// TIA Portal V18 export
DATA_BLOCK "AXIS_Y_Motion_V2_Festo_PtP_Drives_PN_DB"   // DB1
AUTHOR : Festo
FAMILY : E-.Drives
VERSION : 1.5
// stored: AutoNumber true, DBAccessibleFromOPCUA true, InstanceOfName Festo_PtP_Drives_PN, InstanceOfType FB
"Festo_PtP_Drives_PN"
   // VAR_INPUT
   //    ModePos : Int;
   //    EnableAxis : Bool;
   //    CancelTraversing : Bool;
   //    IntermediateStop : Bool;
   //    Positive : Bool;
   //    Negative : Bool;
   //    Jog1 : Bool;
   //    Jog2 : Bool;
   //    AckError : Bool;
   //    ExecuteMode : Bool;
   //    ReleaseBrake : Bool;
   //    TravelToFixStop : Bool;
   //    Position : DInt;
   //    Velocity : DInt;
   //    OverV : Int;
   //    OverAcc : Int;
   //    OverDec : Int;
   //    ConfigEPos : DWord;
   //    BaseSpeedValue : Real;
   //    HardwareId : HW_IO;
   // END_VAR
   // VAR_OUTPUT
   //    AxisEnabled : Bool;
   //    AxisPosOk : Bool;
   //    AxisSpFixed : Bool;
   //    AxisAckSetpoint : Bool;
   //    ClampTorqueReached : Bool;
   //    AxisRef : Bool;
   //    AxisWarn : Bool;
   //    AxisError : Bool;
   //    Lockout : Bool;
   //    ActVelocity : Real;
   //    ActPosition : DInt;
   //    ActMode : Int;
   //    EPosZSW1 : Word;
   //    EPosZSW2 : Word;
   //    ActWarn : Word;
   //    ActFault : Word;
   //    Error : Bool;
   //    Status : Word;
   //    DiagID : Word;
   // END_VAR
   // VAR
   //    stat_Ready4Motion : Bool;
   //    stat_ExecuteIntern : Bool;
   //    stat_StepHome : UInt;
   //    stat_RetDPRD : Int;
   //    stat_RetDPWR : Int;
   //    stat_CycWrite : Struct
   //       STW1 : Struct
   //          jog1 : Bool;
   //          jog2 : Bool;
   //          controlByPlc : Bool;
   //          StartHoming : Bool;
   //          ReleaseBrake : Bool;
   //          ExternalBlockChange : Bool;
   //          reserved14 : Bool;
   //          reserved15 : Bool;
   //          on : Bool;
   //          noCoastStop : Bool;
   //          noQuickStop : Bool;
   //          enableOperation : Bool;
   //          cancelTraversing : Bool;
   //          intermediateStop : Bool;
   //          activateTraversing : Bool;
   //          acknowledgeFault : Bool;
   //       END_STRUCT;
   //       POS_STW1 : Struct
   //          MDI_MOD : Bool;
   //          PosModulo : Bool;
   //          NegModulo : Bool;
   //          reserved11 : Bool;
   //          reserved12 : Bool;
   //          reserved13 : Bool;
   //          SetupMode : Bool;
   //          MDI_Activate : Bool;
   //          travBlockBit0 : Bool;
   //          travBlockBit1 : Bool;
   //          travBlockBit2 : Bool;
   //          travBlockBit3 : Bool;
   //          travBlockBit4 : Bool;
   //          travBlockBit5 : Bool;
   //          travBlockBit6 : Bool;
   //          reserved7 : Bool;
   //       END_STRUCT;
   //       POS_STW2 : Struct
   //          FlyingRef : Bool;
   //          reserved9 : Bool;
   //          SelectProbe : Bool;
   //          ProbeEdgeEval : Bool;
   //          reserved12 : Bool;
   //          reserved13 : Bool;
   //          "SW-Limit" : Bool;
   //          "HW-Limit" : Bool;
   //          Trackingmode : Bool;
   //          SetReferencePoint : Bool;
   //          reserved2 : Bool;
   //          reserved3 : Bool;
   //          reserved4 : Bool;
   //          jog_inc : Bool;
   //          reserved6 : Bool;
   //          reserved7 : Bool;
   //       END_STRUCT;
   //       STW2 : Struct
   //          TravelToFixStop : Bool;
   //          reserved9 : Bool;
   //          reserved10 : Bool;
   //          reserved11 : Bool;
   //          signOfLifeBit0 : Bool;
   //          signOfLifeBit1 : Bool;
   //          signOfLifeBit2 : Bool;
   //          signOfLifeBit3 : Bool;
   //          reserved0 : Bool;
   //          reserved1 : Bool;
   //          reserved2 : Bool;
   //          reserved3 : Bool;
   //          reserved4 : Bool;
   //          reserved5 : Bool;
   //          reserved6 : Bool;
   //          reserved7 : Bool;
   //       END_STRUCT;
   //       Override : Word;
   //       MDI_TARPOS : DInt;
   //       MDI_VELOCITY : DInt;
   //       MDI_ACC : UInt;
   //       MDI_DEC : UInt;
   //       reserved11 : Word;
   //    END_STRUCT;
   //    stat_CycRead : Struct
   //       ZSW1 : Struct
   //          followingErrorInTolerance : Bool;
   //          controlRequest : Bool;
   //          targetPosReached : Bool;
   //          homePosSet : Bool;
   //          acknowledgeTraversingBlockActivated : Bool;
   //          driveStopped : Bool;
   //          axisAccelerates : Bool;
   //          axisDecelerates : Bool;
   //          readyForSwitchOn : Bool;
   //          ready : Bool;
   //          operationEnabled : Bool;
   //          faultPresent : Bool;
   //          noCoastingActive : Bool;
   //          noQuickStopActive : Bool;
   //          switchingOnInhibitedActive : Bool;
   //          warningActive : Bool;
   //       END_STRUCT;
   //       POS_ZSW1 : Word;
   //       POS_ZSW2 : Word;
   //       ZSW2 : Struct
   //          deviceSpecificBit8 : Bool;
   //          deviceSpecificBit9 : Bool;
   //          deviceSpecificBit10 : Bool;
   //          deviceSpecificBit11 : Bool;
   //          doSignOfLifeBit0 : Bool;
   //          doSignOfLifeBit1 : Bool;
   //          doSignOfLifeBit2 : Bool;
   //          doSignOfLifeBit3 : Bool;
   //          deviceSpecificBit0 : Bool;
   //          deviceSpecificBit1 : Bool;
   //          deviceSpecificBit2 : Bool;
   //          deviceSpecificBit3 : Bool;
   //          deviceSpecificBit4 : Bool;
   //          deviceSpecificBit5 : Bool;
   //          deviceSpecificBit6 : Bool;
   //          deviceSpecificBit7 : Bool;
   //       END_STRUCT;
   //       MELDW : Word;
   //       XIST_A : DInt;
   //       NIST_B : DInt;
   //       Fault_Code : Word;
   //       Warn_Code : Word;
   //       Reserved : Word;
   //    END_STRUCT;
   //    stat_ExecAux : Bool;
   //    stat_ExecR_Trig : Bool;
   //    stat_Jog1PAux : Bool;
   //    stat_Jog1PR_trig : Bool;
   //    stat_Jog2PAux : Bool;
   //    stat_Jog2PR_trig : Bool;
   //    stat_Jog1PMode8Aux : Bool;
   //    stat_Jog1PMode8R_trig : Bool;
   //    stat_Jog2PMode8Aux : Bool;
   //    stat_Jog2PMode8R_trig : Bool;
   //    stat_Status : Word;
   //    statStartCounter : Int;
   //    stat_ActMode : Int;
   //    stat_MaxCounterRetries { ExternalAccessible := 'False'; ExternalVisible := 'False'; ExternalWritable := 'False'} : Int;
   // END_VAR
BEGIN
END_DATA_BLOCK
